% RSLogix 500 project TOFF Que 1.RSS, saved by version 8.30.00.15 %
PROJECT "UNTITLED"    % processor: MicroLogix 1400 %

PROGRAM FILES
  LAD 2   4 rungs

DATA FILES
  O0 OUTPUT  6 elements
  I1 INPUT  8 elements
  S2 STATUS  66 elements
  B3 BINARY  1 elements
  T4 TIMER  4 elements
  C5 COUNTER  1 elements
  R6 CONTROL  1 elements
  N7 INTEGER  1 elements
  F8 FLOAT  1 elements

LADDER 2
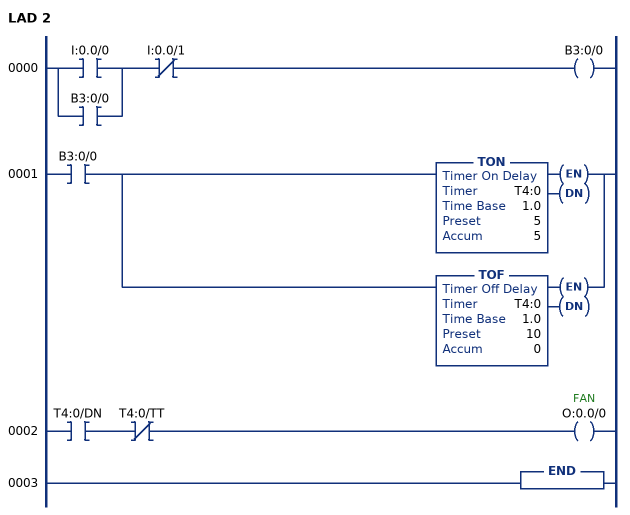
% Rung: 0 %
SOR BST XIC I:0.0/0 NXB XIC B3:0/0 BND XIO I:0.0/1 OTE B3:0/0 EOR
% Rung: 1 %  % edit flag set %
SOR XIC B3:0/0 BST TON T4:0 1.0 5 5 NXB TOF T4:0 1.0 10 0 BND EOR
% Rung: 2 %  % edit flag set %
SOR XIC T4:0/DN XIO T4:0/TT OTE O:0.0/0 EOR
%   O:0.0/0  FAN %
% Rung: 3 %
SOR END EOR

OTHER DOCUMENTED ADDRESSES
  O:0.0/1  MOTOR

DATA TABLE (non-zero values as saved)
DATA B3
% B3:0 % 0X0003
DATA T4
% .PRE .ACC %
% T4:0 % 5 5
% T4:1 % 10 0
% T4:2 % 5 0
% T4:3 % 23 0
